// TIA Portal V17 export
// export: Created 2022-07-28T18:03:17.1027592Z, ExportSetting None, DisplayName Totally Integrated Automation Portal, DisplayVersion V17, DisplayName TIA Portal Openness, DisplayVersion V17, DisplayName TIA Portal Teamcenter Gateway, DisplayVersion V17, DisplayName TIA Portal Version Control Interface, DisplayVersion V17, DisplayName TIA Portal Test Suite Advanced, DisplayVersion V17, DisplayName SINAMICS Startdrive Advanced, DisplayVersion V17, DisplayName SINAMICS DCC, DisplayVersion V17, DisplayName SINAMICS Startdrive G130, G150, S120, S150, SINAMICS MV, S210, DisplayVersion V17, DisplayName SINAMICS Startdrive G110M, G120, G120C, G120D, G120P, G115D, DisplayVersion V17, DisplayName STEP 7 Professional, DisplayVersion V17, DisplayName SIMATIC Energy Suite, DisplayVersion V17, DisplayName STEP 7 CFC, DisplayVersion V17, DisplayName STEP 7 Safety, DisplayVersion V17, DisplayName WinCC Advanced / Unified PC, DisplayVersion V17, DisplayName SIMATIC Visualization Architect, DisplayVersion V17
TYPE "_Inverter_352Tel_CTW_Bits"
   STRUCT
      OFF1 : Bool := false;   // Bit 0 - 0 = Switch-off with ramp-down p1121
      OFF2 : Bool := true;   // Bit 1 - 0 = Switch-off immediately, motor coast to stop
      OFF3 : Bool := true;   // Bit 2 - 0 = Quick stop with ramp-down p1135
      EnableOperation : Bool := true;   // Bit 3 - 1 = Switch-on motor (pulses can be enabled)
      EnableRFG : Bool := true;   // Bit 4 - 1 = Enable ramp-function generator
      FrozeRFG : Bool := true;   // Bit 5 - 0 = Ramp-function generator output is frozen
      EnableSetpoint : Bool := true;   // Bit 6 - 1 = Motor accelerates with ramp p1120; 0 = Motor brakes with ramp p1121
      Acknowlege : Bool;   // Bit 7 - 1 = Acknowlege faults with positive edge. If the ON command still active, the inverter switches to "closing lockout" state
      Bit8_NotUsed : Bool;   // Bit 8 - NU
      Bit9_NotUsed : Bool;   // Bit 9 - NU
      CtrlByPLC : Bool := true;   // Bit 10 - 1 = Control via fieldbus, process data valid
      ChangeDir : Bool;   // Bit 11 - 1 = Change direction. Setpoint is inverted in the drive
      Bit12_NotUsed : Bool;   // Bit 12 - NU
      MOP_Up : Bool;   // Bit 13 - 1 = Motorized potentiometer is increased
      MOP_Dwn : Bool;   // Bit 14 - 1 = Motorized potentiometer is decreased
      Bit15_NotUsed : Bool;   // Bit 15 - NU
   END_STRUCT;
END_TYPE
